ABB RobotStudio station: sesion2_parte2.rspag

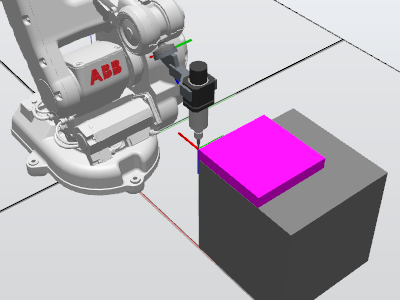
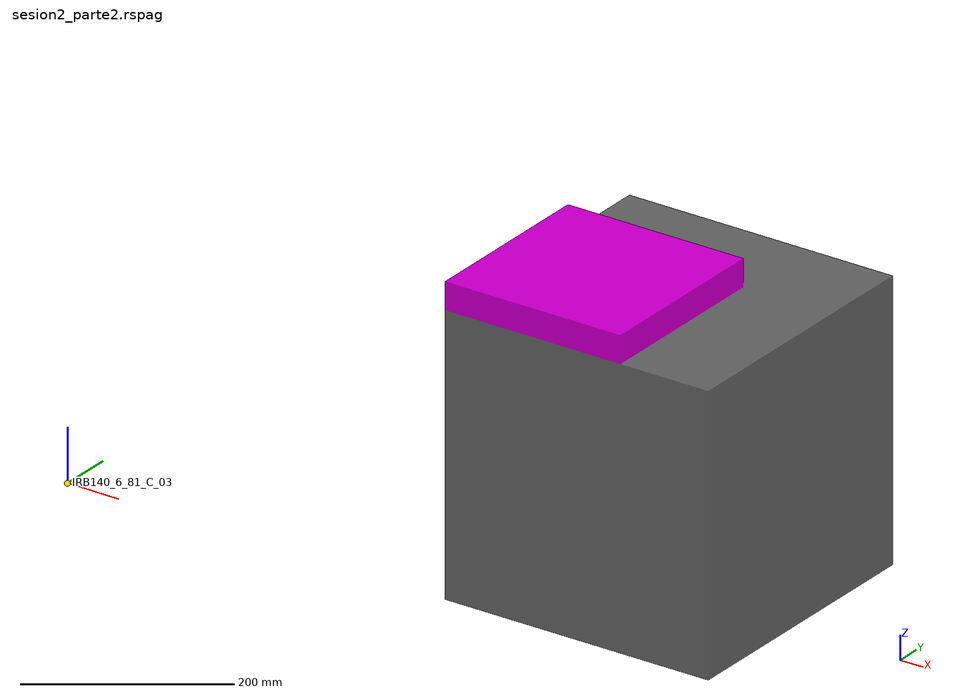
[picture v1: parts stored in the station drawn from their meshes, with robot base, taught points and paths (robot models come from the ABB library and are not in the file)]
--- station ---
Station sesion2 (saved by RobotStudio 24.1.10713.1)
Controller Controlador2
  mechanical unit ROB_1: IRB140_6_81_C_03, 6 joints, base frame (0, 0, 0) mm
Layout (positions relative to the parent item):
  - IRB140_6_81_C_03 [mechanism, from %ABB.RobotStudio.Models.IRB140%\IRB140_6_81_C_G_03.rslib] at (0, 0, 0) mm; joint values [0, -0.4778, 0.7168, 0, 0.6687, 0] (rad or m)
  - MyTool [mechanism, from Training Objects\myTool.rslib] at (313.67, 0, 530.53) mm, rotated rx 180 ry 38 rz 180 deg
  - Pieza_1 [part], size 300 x 300 x 300 mm
  - Pieza_8 [part], size 200 x 200 x 30 mm
Attachment: MyTool is attached to IRB140_6_81_C_03 / Link6
Targets, tools, work objects and paths stored in the station and not in the controller backup, written as RAPID:
! task T_ROB1
MODULE Module1
  PROC Path_10()
    MoveL pIni,v1000,z100,MyTool\WObj:=wobj0;
  ENDPROC
ENDMODULE


--- Backups/Controlador2/RAPID/TASK1/PROGMOD/CalibData.mod ---
MODULE CalibData
    PERS tooldata MyTool:=[TRUE,[[31.792631019,0,229.638935148],[0.945518576,0,0.325568154,0]],[1,[0,0,1],[1,0,0,0],0,0,0]];
ENDMODULE

--- Backups/Controlador2/RAPID/TASK1/PROGMOD/Module1.mod ---
MODULE Module1
        CONST robtarget pIni:=[[430,0,330],[0,0,1,0],[0,0,0,0],[9E+09,9E+09,9E+09,9E+09,9E+09,9E+09]];
!***********************************************************
    !
    ! M?dulo:  Module1
    !
    ! Descripción:
    !   <Introduzca la descripción aquí>
    !
    ! Autor: yisus
    !
    ! Versión: 1.0
    !
    !***********************************************************


    !***********************************************************
    !
    ! Procedimiento Main
    !
    !   Este es el punto de entrada de su programa
    !
    !***********************************************************
    PROC main()
        !Add your code here
        CONST num lado:= 200;
        Cuadrado pIni, lado;
    ENDPROC
    PROC Cuadrado (robtarget pInicial,num  lado)
        VAR robtarget pAux;
        MoveL pInicial,v1000,z100,MyTool\WObj:=wobj0;
        pAux:= Offs(pInicial,lado,0,0);
        MoveL pAux,v1000,z0,MyTool\WObj:=wobj0;
         pAux:= Offs(pInicial,lado,lado,0);
        MoveL pAux,v1000,z0,MyTool\WObj:=wobj0;
         pAux:= Offs(pInicial,0,lado,0);
        MoveL pAux,v1000,z0,MyTool\WObj:=wobj0;
        MoveL pInicial,v1000,z100,MyTool\WObj:=wobj0;
        TPWrite "Cuadrado terminado" ;


    ENDPROC
ENDMODULE
